TM_CircleCmd_Instance(
	Enable:=TM_CircleCmd_Enable,
	Execute:=TM_CircleCmd_Execute,
	RobotID:=ListenNode_Connect_TCP_Socket,
	DataFormat:=TM_CircleCmd_DataFormat,
	ArcPoint:=TM_CircleCmd_ArcPoint,
	EndArcPoint:=TM_CircleCmd_EndArcPoint,
	Speed:=TM_CircleCmd_Speed,
	AccelTime:=TM_CircleCmd_AccelTime,
	Blending:=TM_CircleCmd_Blending,
	ArcAngle:=TM_CircleCmd_ArcAngle,
	PrecisePos:=TM_CircleCmd_PrecisePos,
	Command:=TM_CircleCmd_Command,
	ActivateExit:=TM_CircleCmd_ActivateExit,
	ListenNode:=TM_CircleCmd_ListenNode,
	TimeOut:=T#3600s,
	CommandID:=TM_CircleCmd_CommandID,
	Done=>TM_CircleCmd_Done,
	Busy=>TM_CircleCmd_Busy,
	Error=>TM_CircleCmd_Error,
	ErrorID=>TM_CircleCmd_ErrorID,
	TimeOutET=>TM_CircleCmd_TimeOutET
);

TM_ChangeBase_Instance(
	Enable:=TM_ChangeBase_Enable,
	Execute:=TM_ChangeBase_Execute,
	RobotID:=ListenNode_Connect_TCP_Socket,
	Base:=TM_ChangeBase_Base,
	Command:=TM_ChangeBase_Command,
	ActivateExit:=TM_ChangeBase_ActivateExit,
	ListenNode:=TM_ChangeBase_ListenNode,
	TimeOut:=T#3600s,
	CommandID:=TM_ChangeBase_CommandID,
	Done=>TM_ChangeBase_Done,
	Busy=>TM_ChangeBase_Busy,
	Error=>TM_ChangeBase_Error,
	ErrorID=>TM_ChangeBase_ErrorID,
	TimeOutET=>TM_ChangeBase_TimeOutET
);
END_PROGRAM

PROGRAM CobotModbusComms
VAR
    ButtonStatus : TMmodbus\sRobotStickButtons;
    TM_Modbus : TMmodbus\fbTMmodbus1_80;
    PortIsReady : BOOL;
    test : BOOL;
END_VAR
VAR_EXTERNAL
    StartCommunications : BOOL;
    MBerror : WORD;
    RobotCoordinates : TMmodbus\sRobotCoordinate;  (* Standard robot coordinates *)
    TouchCoordinates : TMmodbus\sRobotCoordinateTouch;  (* Robot coordinates coming from the 'Touch Stop' node. *)
    RobotStatus : TMmodbus\sRobotStatus;
    RobotVitals : TMmodbus\sRobotVitals;
    Config : TMmodbus\sConfiguration;
    RobotTCPLive : TMmodbus\sRobotTCPLive;
    CurrentProjectName : string[200];
    NewProjectName : string[200];
    CommsRoundRobin : REAL;
    TCPerror : WORD;
    RobotControlBoxInfo : TMmodbus\sRobotControllerData;
    Buttons : TMmodbus\sRobotStickButtons;
    RobotIO : TMmodbus\sRobotIO;
    RobotSafetySettings : TMmodbus\sRobotSafety;
    RealsToRobot : ARRAY[0..49] OF real;
    FloatsFromRobot : ARRAY[0..49] OF real;
    BoolsToRobot : ARRAY[0..63] OF BOOL;
    Int16sFromRobot : ARRAY[0..49] OF INT;
    BoolsFromRobot : ARRAY[0..63] OF BOOL;
    IntsToRobot : ARRAY[0..49] OF INT;
    CommunicationsStatus : _eCONNECTION_STATE;
    CommunicationsBusy : BOOL;
    RetryCounter : UINT;
    TCPerrorOriginator : TMModbus\eFunctionBlockError;
    RobotJointTorques : TMmodbus\sRobotJointTorque;
    TaskTimeFB : REAL;
    StartProgram : BOOL;
END_VAR
VAR
    _e1 : R_TRIG;
    _e2 : F_TRIG;
    _p3 : BOOL;
    _e4 : F_TRIG;
END_VAR

(* Section TM12ModbusComms: ladder, written here as Structured Text *)

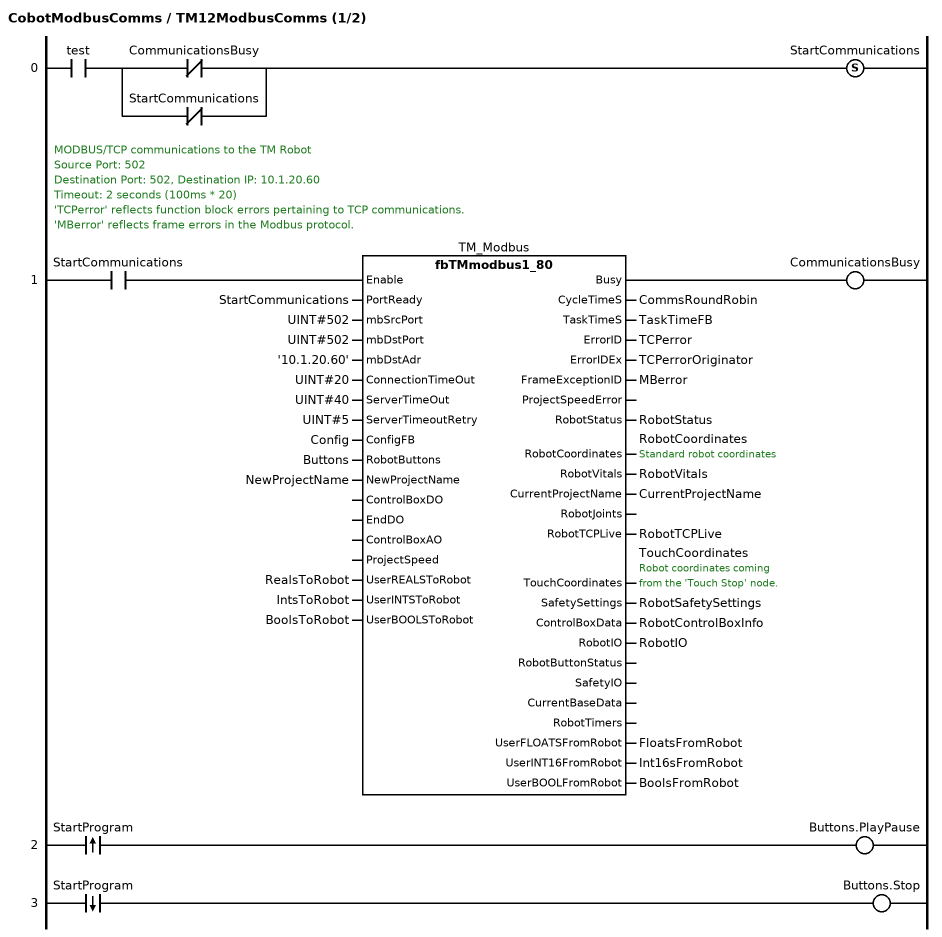
(* Rung 0 *)
IF test AND (NOT CommunicationsBusy OR NOT StartCommunications) THEN StartCommunications := TRUE; END_IF;
(* Rung 1: MODBUS/TCP communications to the TM Robot / Source Port: 502 / Destination Port: 502, Destination IP: 10.1.20.60 / Timeout: 2 seconds (100ms * 20) / 'TCPerror' reflects function block errors pertaining to TCP communications. / 'MBerror' reflects frame errors in the Modbus protocol. *)
TM_Modbus(Enable := StartCommunications, PortReady := StartCommunications, mbSrcPort := UINT#502, mbDstPort := UINT#502, mbDstAdr := '10.1.20.60', ConnectionTimeOut := UINT#20, ServerTimeOut := UINT#40, ServerTimeoutRetry := UINT#5, ConfigFB := Config, RobotButtons := Buttons, NewProjectName := NewProjectName, UserREALSToRobot := RealsToRobot, UserINTSToRobot := IntsToRobot, UserBOOLSToRobot := BoolsToRobot, CycleTimeS => CommsRoundRobin, TaskTimeS => TaskTimeFB, ErrorID => TCPerror, ErrorIDEx => TCPerrorOriginator, FrameExceptionID => MBerror, RobotStatus => RobotStatus, RobotCoordinates => RobotCoordinates, RobotVitals => RobotVitals, CurrentProjectName => CurrentProjectName, RobotTCPLive => RobotTCPLive, TouchCoordinates => TouchCoordinates, SafetySettings => RobotSafetySettings, ControlBoxData => RobotControlBoxInfo, RobotIO => RobotIO, UserFLOATSFromRobot => FloatsFromRobot, UserINT16FromRobot => Int16sFromRobot, UserBOOLFromRobot => BoolsFromRobot);
CommunicationsBusy := TM_Modbus.Busy;
(* Rung 2 *)
_e1(CLK := StartProgram);
Buttons.PlayPause := _e1.Q;
(* Rung 3 *)
_e2(CLK := StartProgram);
Buttons.Stop := _e2.Q;

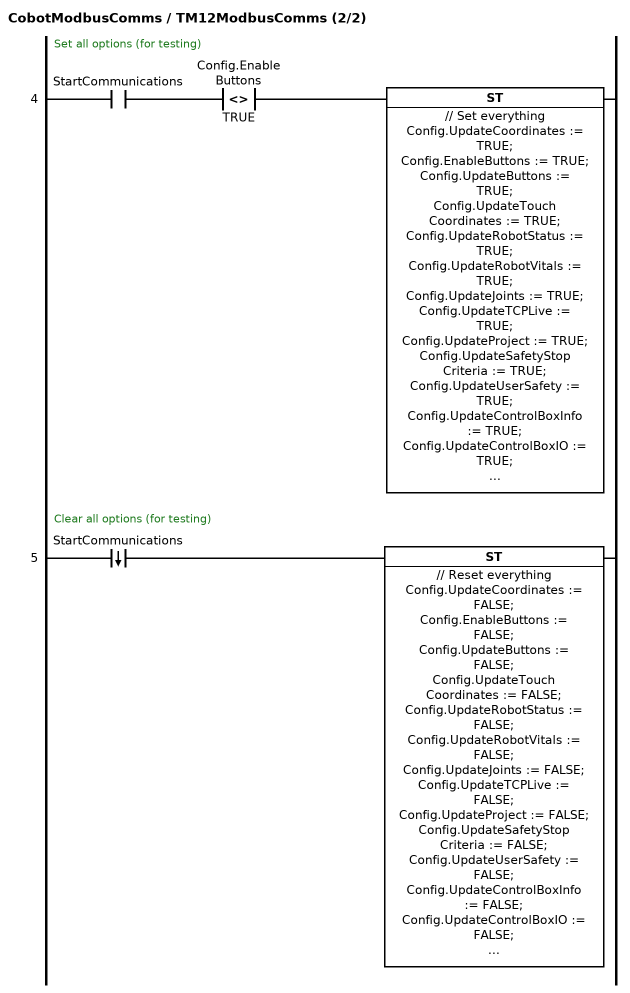
(* Rung 4: Set all options (for testing) *)
_p3 := StartCommunications AND (Config.EnableButtons <> TRUE);
IF _p3 THEN
    // Set everything
    Config.UpdateCoordinates := TRUE;
    Config.EnableButtons := TRUE;
    Config.UpdateButtons := TRUE;
    Config.UpdateTouchCoordinates := TRUE;
    Config.UpdateRobotStatus := TRUE;
    Config.UpdateRobotVitals := TRUE;
    Config.UpdateJoints := TRUE;
    Config.UpdateTCPLive := TRUE;
    Config.UpdateProject := TRUE;
    Config.UpdateSafetyStopCriteria := TRUE;
    Config.UpdateUserSafety := TRUE;
    Config.UpdateControlBoxInfo := TRUE;
    Config.UpdateControlBoxIO := TRUE;
    Config.UpdateEndIO := TRUE;
    Config.UpdateSafetyIO := TRUE;
    Config.UpdateUserFLOATS := TRUE;
    Config.UpdateUserINT16 := TRUE;
    Config.UpdateUserCoils := TRUE;
    Config.EnableControlBoxDO := TRUE;
    Config.EnableControlBoxAO := TRUE;
    Config.EnableEndEffectorDO := TRUE;
    Config.UpdateBase := TRUE;
    Config.UpdateTimers := TRUE;
    Config.EnableSpeedChange := TRUE;
END_IF;
(* Rung 5: Clear all options (for testing) *)
_e4(CLK := StartCommunications);
IF _e4.Q THEN
    // Reset everything
    Config.UpdateCoordinates := FALSE;
    Config.EnableButtons := FALSE;
    Config.UpdateButtons := FALSE;
    Config.UpdateTouchCoordinates := FALSE;
    Config.UpdateRobotStatus := FALSE;
    Config.UpdateRobotVitals := FALSE;
    Config.UpdateJoints := FALSE;
    Config.UpdateTCPLive := FALSE;
    Config.UpdateProject := FALSE;
    Config.UpdateSafetyStopCriteria := FALSE;
    Config.UpdateUserSafety := FALSE;
    Config.UpdateControlBoxInfo := FALSE;
    Config.UpdateControlBoxIO := FALSE;
    Config.UpdateEndIO := FALSE;
    Config.UpdateSafetyIO := FALSE;
    Config.UpdateUserFLOATS := FALSE;
    Config.UpdateUserINT16 := FALSE;
    Config.UpdateUserCoils := FALSE;
    Config.EnableControlBoxDO := FALSE;
    Config.EnableControlBoxAO := FALSE;
    Config.EnableEndEffectorDO := FALSE;
    Config.UpdateBase := FALSE;
    Config.UpdateTimers := FALSE;
    Config.EnableSpeedChange := FALSE;
END_IF;
END_PROGRAM